{attribute 'linkalways'} 
{attribute 'no_explicit_call' := 'This FB is a CLASS and must be accessed using methods or properties'}
{attribute 'enable_dynamic_creation'}
FUNCTION_BLOCK DefaultHomingBuilder IMPLEMENTS I_HomingBuilder, I_PositioningHomingBuilder, I_DefaultHomingBuilder
VAR
	_axis : Axis;
	_position : LREAL;
	_options : ST_HomingOptions;
	_cam : REFERENCE TO BOOL;
END_VAR

METHOD BuildDefaultHomingCommand : HomingCommand
VAR
	pCmd : POINTER TO Mc2HomingCommand;
	cmd : HomingCommand;
END_VAR
pCmd := __NEW(Mc2HomingCommand(
	axis := _axis,
	position := _position,
	mode := HomingMode.Default,
	options := _options,
	cam := _cam
));
BuildDefaultHomingCommand := pCmd^;
END_METHOD

METHOD BuildDirectHomingCommand : HomingCommand
VAR
	pCmd : POINTER TO Mc2HomingCommand;
	cmd : HomingCommand;
	null : BOOL;
END_VAR
pCmd := __NEW(Mc2HomingCommand(
	axis := _axis,
	position := _position,
	mode := HomingMode.Direct,
	options := _options,
	cam := null
));
BuildDirectHomingCommand := pCmd^;
END_METHOD

METHOD BuildForceCalibrationCommand : HomingCommand
VAR
	pCmd : POINTER TO Mc2HomingCommand;
	cmd : HomingCommand;
	null : BOOL;
END_VAR
pCmd := __NEW(Mc2HomingCommand(
	axis := _axis,
	position := _position,
	mode := HomingMode.ForceCalibration,
	options := _options,
	cam := null
));
BuildForceCalibrationCommand := pCmd^;
END_METHOD

METHOD BuildResetCalibrationCommand : HomingCommand
VAR
	pCmd : POINTER TO Mc2HomingCommand;
	cmd : HomingCommand;
	null : BOOL;
END_VAR
pCmd := __NEW(Mc2HomingCommand(
	axis := _axis,
	position := _position,
	mode := HomingMode.ResetCalibration,
	options := _options,
	cam := null
));
BuildResetCalibrationCommand := pCmd^;
END_METHOD

METHOD Cam : I_DefaultHomingBuilder
VAR_INPUT
	value : REFERENCE TO BOOL;
END_VAR
_cam REF= value;
Cam := THIS^;
END_METHOD

METHOD ClearLag : I_PositioningHomingBuilder
_options.ClearPositionLag := TRUE;
ClearLag := THIS^;
END_METHOD

METHOD FB_init : BOOL
VAR_INPUT
	bInitRetains : BOOL; // if TRUE, the retain variables are initialized (warm start / cold start)
	bInCopyCode : BOOL;  // if TRUE, the instance afterwards gets moved into the copy code (online change)
	axis : Axis;
END_VAR
_axis := axis;
END_METHOD

METHOD KeepLag : I_PositioningHomingBuilder
_options.ClearPositionLag := FALSE;
KeepLag := THIS^;
END_METHOD

METHOD Position : I_PositioningHomingBuilder
VAR_INPUT
	value : LREAL;
END_VAR
_position := value;
Position := THIS^;
END_METHOD

METHOD ReferenceMode : I_DefaultHomingBuilder
VAR_INPUT
	value : EncoderReferenceMode;
END_VAR
_options.ReferenceMode := value;
ReferenceMode := THIS^;
END_METHOD

METHOD SearchDirection : I_DefaultHomingBuilder
VAR_INPUT
	value : Direction;
END_VAR
_options.SearchDirection := value;
SearchDirection := THIS^;
END_METHOD

METHOD SearchVelocity : I_DefaultHomingBuilder
VAR_INPUT
	value	: LREAL;
END_VAR
_options.SearchVelocity := value;
SearchVelocity := THIS^;
END_METHOD

METHOD SyncDirection : I_DefaultHomingBuilder
VAR_INPUT
	value : Direction;
END_VAR
_options.SyncDirection := value;
SyncDirection := THIS^;
END_METHOD

METHOD SyncVelocity : I_DefaultHomingBuilder
VAR_INPUT
	value : LREAL;
END_VAR
_options.SyncVelocity := value;
SyncVelocity := THIS^;
END_METHOD

END_FUNCTION_BLOCK

(* stored: Version 1.1.0.1, ProductVersion 3.1.4026.13
   POU DefaultHomingBuilder: Id {69109941-4397-0e86-12a8-1287758a9f8c}, SpecialFunc None
   Folder Builders: Id {088d206f-dadb-0b80-0602-4837e014254b}
   Folder Property Setters: Id {fb6f9a3c-7c86-012f-1f8f-44e6795c4fb6}
   Method BuildDefaultHomingCommand: Id {ddf6d26a-c270-0244-0b05-cc1fe38b015a}
   Method BuildDirectHomingCommand: Id {0538d939-3623-0bef-1dc3-ec51bfc7c90b}
   Method BuildForceCalibrationCommand: Id {f211545c-7420-0fdd-3498-6a4327f8f598}
   Method BuildResetCalibrationCommand: Id {38a7edc9-6421-03eb-16dc-1573f361dd71}
   Method Cam: Id {9c6c92ab-bf2f-0077-035d-a8caeebd0c13}
   Method ClearLag: Id {cfabbc72-1c7a-00cd-10ab-c1323fe10789}
   Method FB_init: Id {c64a5780-0a7b-0f4c-009e-2e6055b4ae84}
   Method KeepLag: Id {176d099b-7a1f-0873-0349-a879c2bd2c88}
   Method Position: Id {cf3da0f8-3163-0786-12ba-003db5badef3}
   Method ReferenceMode: Id {179e90f9-3718-0e96-01a6-1e8c9462942e}
   Method SearchDirection: Id {6a808f82-fe2a-0ac5-3e42-ae84fad4ad51}
   Method SearchVelocity: Id {b5f05c0d-3711-0e12-0c2e-504330470664}
   Method SyncDirection: Id {8aa5d5ce-d5db-0d08-0a14-cf73438fe9e0}
   Method SyncVelocity: Id {12319474-f11b-0da2-28b1-30f4db56f1cd} *)
